// TIA Portal V17 export
// export: Created 2024-10-09T16:19:46.1936447Z, ExportSetting WithDefaults, DisplayName Totally Integrated Automation Portal, DisplayVersion V17, DisplayName TIA Portal Openness, DisplayVersion V17, DisplayName TIA Portal Version Control Interface, DisplayVersion V17, DisplayName STEP 7 Professional, DisplayVersion V17, DisplayName STEP 7 Safety, DisplayVersion V17, DisplayName WinCC Advanced, DisplayVersion V17
VAR_GLOBAL   // PLC tag table "Inputs"
   mpDIs AT %I18.0 : "typeMainPanelDI";
   mpAIs AT %I76.0 : "typeMainPanelAI";
   deckAIs AT %I68.0 : "typeDeckControlAI";
   deckDIs AT %I30.0 : "typeDeckControlDI";
   mpCnts AT %I1000.0 : "typeMainPanelCounters";
   whAIs AT %I84.0 : "typeWheelHouseAI";
   whDIs AT %I92.0 : "typeWheelHouseDI";
   driveIn AT %IW94 : Hw_Io;   // start address of ACS800 drive profibus input area
   driveOut AT %QW82 : Hw_Io;   // start address of ACS800 drive profibus output area
END_VAR
